// TIA Portal V20 export
FUNCTION_BLOCK "Simulation"   // FB100, LAD
// stored: MemoryReserve 100, Namespace Unit1.Em2, SetENOAutomatically false
   VAR
      Simulation_addon_Instance { S7_SetPoint := 'True'} : "Simulation_addon";
      Simulation_addon_Instance_1 { S7_SetPoint := 'True'} : "Simulation_addon";
      Simulation_addon_Instance_2 { S7_SetPoint := 'True'} : "Simulation_addon";
      Simulation_addon_Instance_3 { S7_SetPoint := 'True'} : "Simulation_addon";
      Simulation_addon_Instance_4 { S7_SetPoint := 'True'} : "Simulation_addon";
      Simulation_addon_Instance_5 { S7_SetPoint := 'True'} : "Simulation_addon";
      Simulation_addon_Instance_6 { S7_SetPoint := 'True'} : "Simulation_addon";
      Simulation_addon_Instance_7 { S7_SetPoint := 'True'} : "Simulation_addon";
      Simulation_addon_Instance_8 { S7_SetPoint := 'True'} : "Simulation_addon";
      Simulation_addon_Instance_9 { S7_SetPoint := 'True'} : "Simulation_addon";
      Simulation_addon_Instance_10 { S7_SetPoint := 'True'} : "Simulation_addon";
      Simulation_addon_Instance_11 { S7_SetPoint := 'True'} : "Simulation_addon";
      Simulation_addon_Instance_12 { S7_SetPoint := 'True'} : "Simulation_addon";
      Simulation_addon_Instance_13 { S7_SetPoint := 'True'} : "Simulation_addon";
      Simulation_addon_Instance_14 { S7_SetPoint := 'True'} : "Simulation_addon";
      Simulation_addon_Instance_15 { S7_SetPoint := 'True'} : "Simulation_addon";
      Simulation_addon_Instance_16 { S7_SetPoint := 'True'} : "Simulation_addon";
      Simulation_addon_Instance_17 { S7_SetPoint := 'True'} : "Simulation_addon";
      Simulation_addon_Instance_18 { S7_SetPoint := 'True'} : "Simulation_addon";
      Simulation_addon_Instance_19 { S7_SetPoint := 'True'} : "Simulation_addon";
      Simulation_addon_Instance_20 { S7_SetPoint := 'True'} : "Simulation_addon";
      Simulation_addon_Instance_21 { S7_SetPoint := 'True'} : "Simulation_addon";
   END_VAR
BEGIN

REGION Network 1: cmElectrodeFixRightTopFwdBwd
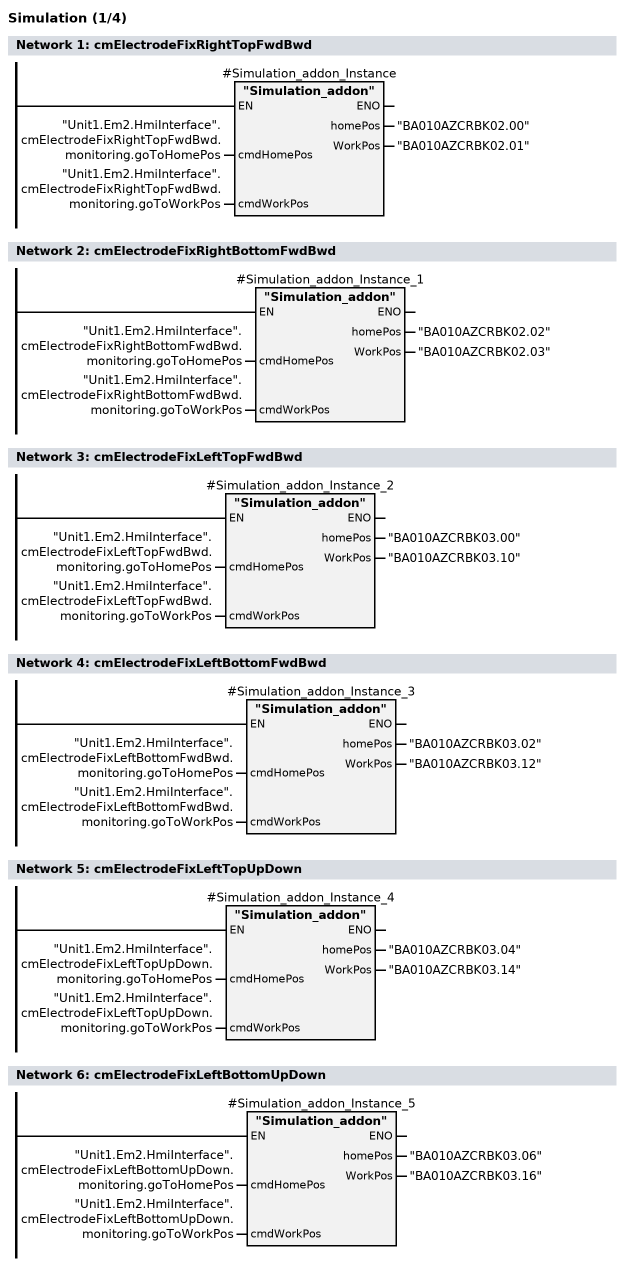
   RUNG wire#powerrail
      #Simulation_addon_Instance(cmdHomePos := "Unit1.Em2.HmiInterface".cmElectrodeFixRightTopFwdBwd.monitoring.goToHomePos, cmdWorkPos := "Unit1.Em2.HmiInterface".cmElectrodeFixRightTopFwdBwd.monitoring.goToWorkPos, homePos => "BA010AZCRBK02.00", WorkPos => "BA010AZCRBK02.01")
   END_RUNG
   // the same network as SCL:
   #Simulation_addon_Instance(cmdHomePos := "Unit1.Em2.HmiInterface".cmElectrodeFixRightTopFwdBwd.monitoring.goToHomePos,   // "Simulation_addon"
                           cmdWorkPos := "Unit1.Em2.HmiInterface".cmElectrodeFixRightTopFwdBwd.monitoring.goToWorkPos,
                           homePos => "BA010AZCRBK02.00",
                           WorkPos => "BA010AZCRBK02.01");
END_REGION

REGION Network 2: cmElectrodeFixRightBottomFwdBwd
   RUNG wire#powerrail
      #Simulation_addon_Instance_1(cmdHomePos := "Unit1.Em2.HmiInterface".cmElectrodeFixRightBottomFwdBwd.monitoring.goToHomePos, cmdWorkPos := "Unit1.Em2.HmiInterface".cmElectrodeFixRightBottomFwdBwd.monitoring.goToWorkPos, homePos => "BA010AZCRBK02.02", WorkPos => "BA010AZCRBK02.03")
   END_RUNG
   // the same network as SCL:
   #Simulation_addon_Instance_1(cmdHomePos := "Unit1.Em2.HmiInterface".cmElectrodeFixRightBottomFwdBwd.monitoring.goToHomePos,   // "Simulation_addon"
                           cmdWorkPos := "Unit1.Em2.HmiInterface".cmElectrodeFixRightBottomFwdBwd.monitoring.goToWorkPos,
                           homePos => "BA010AZCRBK02.02",
                           WorkPos => "BA010AZCRBK02.03");
END_REGION

REGION Network 3: cmElectrodeFixLeftTopFwdBwd
   RUNG wire#powerrail
      #Simulation_addon_Instance_2(cmdHomePos := "Unit1.Em2.HmiInterface".cmElectrodeFixLeftTopFwdBwd.monitoring.goToHomePos, cmdWorkPos := "Unit1.Em2.HmiInterface".cmElectrodeFixLeftTopFwdBwd.monitoring.goToWorkPos, homePos => "BA010AZCRBK03.00", WorkPos => "BA010AZCRBK03.10")
   END_RUNG
   // the same network as SCL:
   #Simulation_addon_Instance_2(cmdHomePos := "Unit1.Em2.HmiInterface".cmElectrodeFixLeftTopFwdBwd.monitoring.goToHomePos,   // "Simulation_addon"
                           cmdWorkPos := "Unit1.Em2.HmiInterface".cmElectrodeFixLeftTopFwdBwd.monitoring.goToWorkPos,
                           homePos => "BA010AZCRBK03.00",
                           WorkPos => "BA010AZCRBK03.10");
END_REGION

REGION Network 4: cmElectrodeFixLeftBottomFwdBwd
   RUNG wire#powerrail
      #Simulation_addon_Instance_3(cmdHomePos := "Unit1.Em2.HmiInterface".cmElectrodeFixLeftBottomFwdBwd.monitoring.goToHomePos, cmdWorkPos := "Unit1.Em2.HmiInterface".cmElectrodeFixLeftBottomFwdBwd.monitoring.goToWorkPos, homePos => "BA010AZCRBK03.02", WorkPos => "BA010AZCRBK03.12")
   END_RUNG
   // the same network as SCL:
   #Simulation_addon_Instance_3(cmdHomePos := "Unit1.Em2.HmiInterface".cmElectrodeFixLeftBottomFwdBwd.monitoring.goToHomePos,   // "Simulation_addon"
                           cmdWorkPos := "Unit1.Em2.HmiInterface".cmElectrodeFixLeftBottomFwdBwd.monitoring.goToWorkPos,
                           homePos => "BA010AZCRBK03.02",
                           WorkPos => "BA010AZCRBK03.12");
END_REGION

REGION Network 5: cmElectrodeFixLeftTopUpDown
   RUNG wire#powerrail
      #Simulation_addon_Instance_4(cmdHomePos := "Unit1.Em2.HmiInterface".cmElectrodeFixLeftTopUpDown.monitoring.goToHomePos, cmdWorkPos := "Unit1.Em2.HmiInterface".cmElectrodeFixLeftTopUpDown.monitoring.goToWorkPos, homePos => "BA010AZCRBK03.04", WorkPos => "BA010AZCRBK03.14")
   END_RUNG
   // the same network as SCL:
   #Simulation_addon_Instance_4(cmdHomePos := "Unit1.Em2.HmiInterface".cmElectrodeFixLeftTopUpDown.monitoring.goToHomePos,   // "Simulation_addon"
                           cmdWorkPos := "Unit1.Em2.HmiInterface".cmElectrodeFixLeftTopUpDown.monitoring.goToWorkPos,
                           homePos => "BA010AZCRBK03.04",
                           WorkPos => "BA010AZCRBK03.14");
END_REGION

REGION Network 6: cmElectrodeFixLeftBottomUpDown
   RUNG wire#powerrail
      #Simulation_addon_Instance_5(cmdHomePos := "Unit1.Em2.HmiInterface".cmElectrodeFixLeftBottomUpDown.monitoring.goToHomePos, cmdWorkPos := "Unit1.Em2.HmiInterface".cmElectrodeFixLeftBottomUpDown.monitoring.goToWorkPos, homePos => "BA010AZCRBK03.06", WorkPos => "BA010AZCRBK03.16")
   END_RUNG
   // the same network as SCL:
   #Simulation_addon_Instance_5(cmdHomePos := "Unit1.Em2.HmiInterface".cmElectrodeFixLeftBottomUpDown.monitoring.goToHomePos,   // "Simulation_addon"
                           cmdWorkPos := "Unit1.Em2.HmiInterface".cmElectrodeFixLeftBottomUpDown.monitoring.goToWorkPos,
                           homePos => "BA010AZCRBK03.06",
                           WorkPos => "BA010AZCRBK03.16");
END_REGION

REGION Network 7: cmUwSemiSplicerVacuumRightTopOnOff
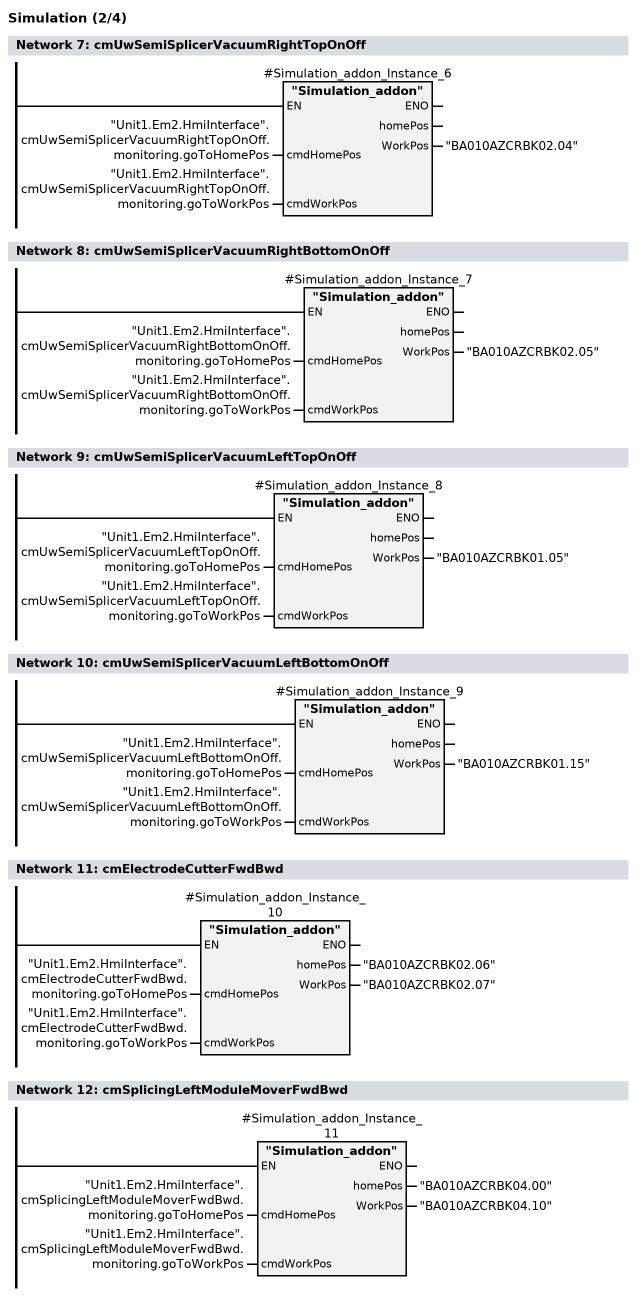
   RUNG wire#powerrail
      #Simulation_addon_Instance_6(cmdHomePos := "Unit1.Em2.HmiInterface".cmUwSemiSplicerVacuumRightTopOnOff.monitoring.goToHomePos, cmdWorkPos := "Unit1.Em2.HmiInterface".cmUwSemiSplicerVacuumRightTopOnOff.monitoring.goToWorkPos, homePos =>, WorkPos => "BA010AZCRBK02.04")
   END_RUNG
   // the same network as SCL:
   #Simulation_addon_Instance_6(cmdHomePos := "Unit1.Em2.HmiInterface".cmUwSemiSplicerVacuumRightTopOnOff.monitoring.goToHomePos,   // "Simulation_addon"
                           cmdWorkPos := "Unit1.Em2.HmiInterface".cmUwSemiSplicerVacuumRightTopOnOff.monitoring.goToWorkPos,
                           WorkPos => "BA010AZCRBK02.04");
END_REGION

REGION Network 8: cmUwSemiSplicerVacuumRightBottomOnOff
   RUNG wire#powerrail
      #Simulation_addon_Instance_7(cmdHomePos := "Unit1.Em2.HmiInterface".cmUwSemiSplicerVacuumRightBottomOnOff.monitoring.goToHomePos, cmdWorkPos := "Unit1.Em2.HmiInterface".cmUwSemiSplicerVacuumRightBottomOnOff.monitoring.goToWorkPos, homePos =>, WorkPos => "BA010AZCRBK02.05")
   END_RUNG
   // the same network as SCL:
   #Simulation_addon_Instance_7(cmdHomePos := "Unit1.Em2.HmiInterface".cmUwSemiSplicerVacuumRightBottomOnOff.monitoring.goToHomePos,   // "Simulation_addon"
                           cmdWorkPos := "Unit1.Em2.HmiInterface".cmUwSemiSplicerVacuumRightBottomOnOff.monitoring.goToWorkPos,
                           WorkPos => "BA010AZCRBK02.05");
END_REGION

REGION Network 9: cmUwSemiSplicerVacuumLeftTopOnOff
   RUNG wire#powerrail
      #Simulation_addon_Instance_8(cmdHomePos := "Unit1.Em2.HmiInterface".cmUwSemiSplicerVacuumLeftTopOnOff.monitoring.goToHomePos, cmdWorkPos := "Unit1.Em2.HmiInterface".cmUwSemiSplicerVacuumLeftTopOnOff.monitoring.goToWorkPos, homePos =>, WorkPos => "BA010AZCRBK01.05")
   END_RUNG
   // the same network as SCL:
   #Simulation_addon_Instance_8(cmdHomePos := "Unit1.Em2.HmiInterface".cmUwSemiSplicerVacuumLeftTopOnOff.monitoring.goToHomePos,   // "Simulation_addon"
                           cmdWorkPos := "Unit1.Em2.HmiInterface".cmUwSemiSplicerVacuumLeftTopOnOff.monitoring.goToWorkPos,
                           WorkPos => "BA010AZCRBK01.05");
END_REGION

REGION Network 10: cmUwSemiSplicerVacuumLeftBottomOnOff
   RUNG wire#powerrail
      #Simulation_addon_Instance_9(cmdHomePos := "Unit1.Em2.HmiInterface".cmUwSemiSplicerVacuumLeftBottomOnOff.monitoring.goToHomePos, cmdWorkPos := "Unit1.Em2.HmiInterface".cmUwSemiSplicerVacuumLeftBottomOnOff.monitoring.goToWorkPos, homePos =>, WorkPos => "BA010AZCRBK01.15")
   END_RUNG
   // the same network as SCL:
   #Simulation_addon_Instance_9(cmdHomePos := "Unit1.Em2.HmiInterface".cmUwSemiSplicerVacuumLeftBottomOnOff.monitoring.goToHomePos,   // "Simulation_addon"
                           cmdWorkPos := "Unit1.Em2.HmiInterface".cmUwSemiSplicerVacuumLeftBottomOnOff.monitoring.goToWorkPos,
                           WorkPos => "BA010AZCRBK01.15");
END_REGION

REGION Network 11: cmElectrodeCutterFwdBwd
   RUNG wire#powerrail
      #Simulation_addon_Instance_10(cmdHomePos := "Unit1.Em2.HmiInterface".cmElectrodeCutterFwdBwd.monitoring.goToHomePos, cmdWorkPos := "Unit1.Em2.HmiInterface".cmElectrodeCutterFwdBwd.monitoring.goToWorkPos, homePos => "BA010AZCRBK02.06", WorkPos => "BA010AZCRBK02.07")
   END_RUNG
   // the same network as SCL:
   #Simulation_addon_Instance_10(cmdHomePos := "Unit1.Em2.HmiInterface".cmElectrodeCutterFwdBwd.monitoring.goToHomePos,   // "Simulation_addon"
                           cmdWorkPos := "Unit1.Em2.HmiInterface".cmElectrodeCutterFwdBwd.monitoring.goToWorkPos,
                           homePos => "BA010AZCRBK02.06",
                           WorkPos => "BA010AZCRBK02.07");
END_REGION

REGION Network 12: cmSplicingLeftModuleMoverFwdBwd
   RUNG wire#powerrail
      #Simulation_addon_Instance_11(cmdHomePos := "Unit1.Em2.HmiInterface".cmSplicingLeftModuleMoverFwdBwd.monitoring.goToHomePos, cmdWorkPos := "Unit1.Em2.HmiInterface".cmSplicingLeftModuleMoverFwdBwd.monitoring.goToWorkPos, homePos => "BA010AZCRBK04.00", WorkPos => "BA010AZCRBK04.10")
   END_RUNG
   // the same network as SCL:
   #Simulation_addon_Instance_11(cmdHomePos := "Unit1.Em2.HmiInterface".cmSplicingLeftModuleMoverFwdBwd.monitoring.goToHomePos,   // "Simulation_addon"
                           cmdWorkPos := "Unit1.Em2.HmiInterface".cmSplicingLeftModuleMoverFwdBwd.monitoring.goToWorkPos,
                           homePos => "BA010AZCRBK04.00",
                           WorkPos => "BA010AZCRBK04.10");
END_REGION

REGION Network 13: cmSplicingRightModuleMoverFwdBwd
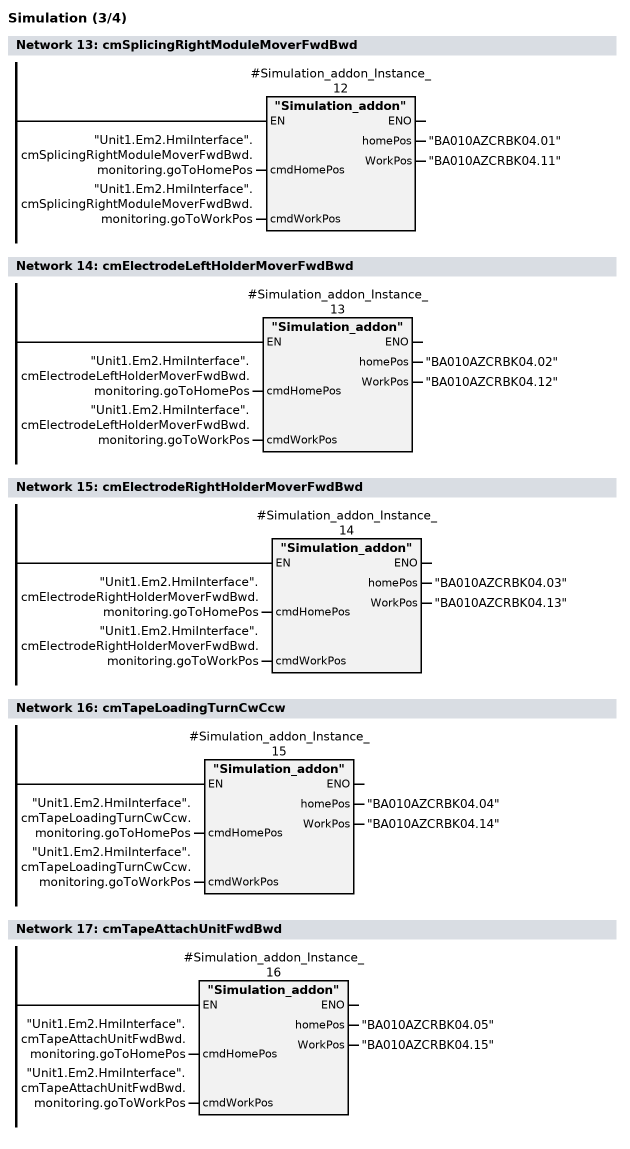
   RUNG wire#powerrail
      #Simulation_addon_Instance_12(cmdHomePos := "Unit1.Em2.HmiInterface".cmSplicingRightModuleMoverFwdBwd.monitoring.goToHomePos, cmdWorkPos := "Unit1.Em2.HmiInterface".cmSplicingRightModuleMoverFwdBwd.monitoring.goToWorkPos, homePos => "BA010AZCRBK04.01", WorkPos => "BA010AZCRBK04.11")
   END_RUNG
   // the same network as SCL:
   #Simulation_addon_Instance_12(cmdHomePos := "Unit1.Em2.HmiInterface".cmSplicingRightModuleMoverFwdBwd.monitoring.goToHomePos,   // "Simulation_addon"
                           cmdWorkPos := "Unit1.Em2.HmiInterface".cmSplicingRightModuleMoverFwdBwd.monitoring.goToWorkPos,
                           homePos => "BA010AZCRBK04.01",
                           WorkPos => "BA010AZCRBK04.11");
END_REGION

REGION Network 14: cmElectrodeLeftHolderMoverFwdBwd
   RUNG wire#powerrail
      #Simulation_addon_Instance_13(cmdHomePos := "Unit1.Em2.HmiInterface".cmElectrodeLeftHolderMoverFwdBwd.monitoring.goToHomePos, cmdWorkPos := "Unit1.Em2.HmiInterface".cmElectrodeLeftHolderMoverFwdBwd.monitoring.goToWorkPos, homePos => "BA010AZCRBK04.02", WorkPos => "BA010AZCRBK04.12")
   END_RUNG
   // the same network as SCL:
   #Simulation_addon_Instance_13(cmdHomePos := "Unit1.Em2.HmiInterface".cmElectrodeLeftHolderMoverFwdBwd.monitoring.goToHomePos,   // "Simulation_addon"
                           cmdWorkPos := "Unit1.Em2.HmiInterface".cmElectrodeLeftHolderMoverFwdBwd.monitoring.goToWorkPos,
                           homePos => "BA010AZCRBK04.02",
                           WorkPos => "BA010AZCRBK04.12");
END_REGION

REGION Network 15: cmElectrodeRightHolderMoverFwdBwd
   RUNG wire#powerrail
      #Simulation_addon_Instance_14(cmdHomePos := "Unit1.Em2.HmiInterface".cmElectrodeRightHolderMoverFwdBwd.monitoring.goToHomePos, cmdWorkPos := "Unit1.Em2.HmiInterface".cmElectrodeRightHolderMoverFwdBwd.monitoring.goToWorkPos, homePos => "BA010AZCRBK04.03", WorkPos => "BA010AZCRBK04.13")
   END_RUNG
   // the same network as SCL:
   #Simulation_addon_Instance_14(cmdHomePos := "Unit1.Em2.HmiInterface".cmElectrodeRightHolderMoverFwdBwd.monitoring.goToHomePos,   // "Simulation_addon"
                           cmdWorkPos := "Unit1.Em2.HmiInterface".cmElectrodeRightHolderMoverFwdBwd.monitoring.goToWorkPos,
                           homePos => "BA010AZCRBK04.03",
                           WorkPos => "BA010AZCRBK04.13");
END_REGION

REGION Network 16: cmTapeLoadingTurnCwCcw
   RUNG wire#powerrail
      #Simulation_addon_Instance_15(cmdHomePos := "Unit1.Em2.HmiInterface".cmTapeLoadingTurnCwCcw.monitoring.goToHomePos, cmdWorkPos := "Unit1.Em2.HmiInterface".cmTapeLoadingTurnCwCcw.monitoring.goToWorkPos, homePos => "BA010AZCRBK04.04", WorkPos => "BA010AZCRBK04.14")
   END_RUNG
   // the same network as SCL:
   #Simulation_addon_Instance_15(cmdHomePos := "Unit1.Em2.HmiInterface".cmTapeLoadingTurnCwCcw.monitoring.goToHomePos,   // "Simulation_addon"
                           cmdWorkPos := "Unit1.Em2.HmiInterface".cmTapeLoadingTurnCwCcw.monitoring.goToWorkPos,
                           homePos => "BA010AZCRBK04.04",
                           WorkPos => "BA010AZCRBK04.14");
END_REGION

REGION Network 17: cmTapeAttachUnitFwdBwd
   RUNG wire#powerrail
      #Simulation_addon_Instance_16(cmdHomePos := "Unit1.Em2.HmiInterface".cmTapeAttachUnitFwdBwd.monitoring.goToHomePos, cmdWorkPos := "Unit1.Em2.HmiInterface".cmTapeAttachUnitFwdBwd.monitoring.goToWorkPos, homePos => "BA010AZCRBK04.05", WorkPos => "BA010AZCRBK04.15")
   END_RUNG
   // the same network as SCL:
   #Simulation_addon_Instance_16(cmdHomePos := "Unit1.Em2.HmiInterface".cmTapeAttachUnitFwdBwd.monitoring.goToHomePos,   // "Simulation_addon"
                           cmdWorkPos := "Unit1.Em2.HmiInterface".cmTapeAttachUnitFwdBwd.monitoring.goToWorkPos,
                           homePos => "BA010AZCRBK04.05",
                           WorkPos => "BA010AZCRBK04.15");
END_REGION

REGION Network 18: SemiSplicerTapeVacuumOnOff
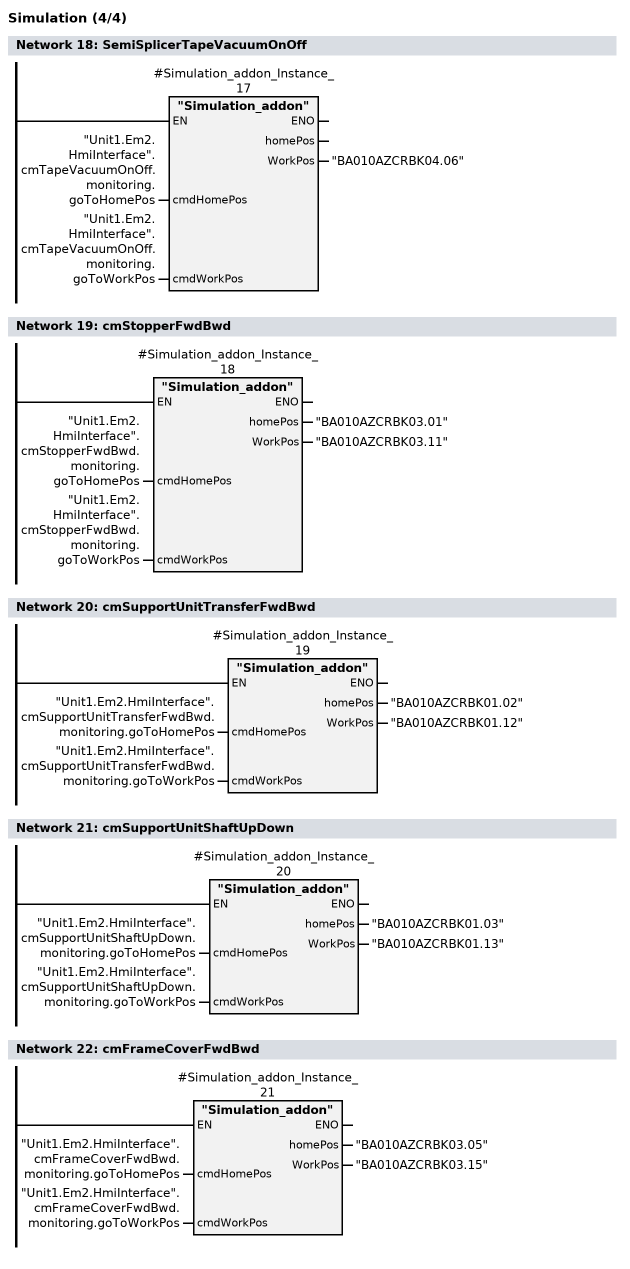
   RUNG wire#powerrail
      #Simulation_addon_Instance_17(cmdHomePos := "Unit1.Em2.HmiInterface".cmTapeVacuumOnOff.monitoring.goToHomePos, cmdWorkPos := "Unit1.Em2.HmiInterface".cmTapeVacuumOnOff.monitoring.goToWorkPos, homePos =>, WorkPos => "BA010AZCRBK04.06")
   END_RUNG
   // the same network as SCL:
   #Simulation_addon_Instance_17(cmdHomePos := "Unit1.Em2.HmiInterface".cmTapeVacuumOnOff.monitoring.goToHomePos,   // "Simulation_addon"
                           cmdWorkPos := "Unit1.Em2.HmiInterface".cmTapeVacuumOnOff.monitoring.goToWorkPos,
                           WorkPos => "BA010AZCRBK04.06");
END_REGION

REGION Network 19: cmStopperFwdBwd
   RUNG wire#powerrail
      #Simulation_addon_Instance_18(cmdHomePos := "Unit1.Em2.HmiInterface".cmStopperFwdBwd.monitoring.goToHomePos, cmdWorkPos := "Unit1.Em2.HmiInterface".cmStopperFwdBwd.monitoring.goToWorkPos, homePos => "BA010AZCRBK03.01", WorkPos => "BA010AZCRBK03.11")
   END_RUNG
   // the same network as SCL:
   #Simulation_addon_Instance_18(cmdHomePos := "Unit1.Em2.HmiInterface".cmStopperFwdBwd.monitoring.goToHomePos,   // "Simulation_addon"
                           cmdWorkPos := "Unit1.Em2.HmiInterface".cmStopperFwdBwd.monitoring.goToWorkPos,
                           homePos => "BA010AZCRBK03.01",
                           WorkPos => "BA010AZCRBK03.11");
END_REGION

REGION Network 20: cmSupportUnitTransferFwdBwd
   RUNG wire#powerrail
      #Simulation_addon_Instance_19(cmdHomePos := "Unit1.Em2.HmiInterface".cmSupportUnitTransferFwdBwd.monitoring.goToHomePos, cmdWorkPos := "Unit1.Em2.HmiInterface".cmSupportUnitTransferFwdBwd.monitoring.goToWorkPos, homePos => "BA010AZCRBK01.02", WorkPos => "BA010AZCRBK01.12")
   END_RUNG
   // the same network as SCL:
   #Simulation_addon_Instance_19(cmdHomePos := "Unit1.Em2.HmiInterface".cmSupportUnitTransferFwdBwd.monitoring.goToHomePos,   // "Simulation_addon"
                           cmdWorkPos := "Unit1.Em2.HmiInterface".cmSupportUnitTransferFwdBwd.monitoring.goToWorkPos,
                           homePos => "BA010AZCRBK01.02",
                           WorkPos => "BA010AZCRBK01.12");
END_REGION

REGION Network 21: cmSupportUnitShaftUpDown
   RUNG wire#powerrail
      #Simulation_addon_Instance_20(cmdHomePos := "Unit1.Em2.HmiInterface".cmSupportUnitShaftUpDown.monitoring.goToHomePos, cmdWorkPos := "Unit1.Em2.HmiInterface".cmSupportUnitShaftUpDown.monitoring.goToWorkPos, homePos => "BA010AZCRBK01.03", WorkPos => "BA010AZCRBK01.13")
   END_RUNG
   // the same network as SCL:
   #Simulation_addon_Instance_20(cmdHomePos := "Unit1.Em2.HmiInterface".cmSupportUnitShaftUpDown.monitoring.goToHomePos,   // "Simulation_addon"
                           cmdWorkPos := "Unit1.Em2.HmiInterface".cmSupportUnitShaftUpDown.monitoring.goToWorkPos,
                           homePos => "BA010AZCRBK01.03",
                           WorkPos => "BA010AZCRBK01.13");
END_REGION

REGION Network 22: cmFrameCoverFwdBwd
   RUNG wire#powerrail
      #Simulation_addon_Instance_21(cmdHomePos := "Unit1.Em2.HmiInterface".cmFrameCoverFwdBwd.monitoring.goToHomePos, cmdWorkPos := "Unit1.Em2.HmiInterface".cmFrameCoverFwdBwd.monitoring.goToWorkPos, homePos => "BA010AZCRBK03.05", WorkPos => "BA010AZCRBK03.15")
   END_RUNG
   // the same network as SCL:
   #Simulation_addon_Instance_21(cmdHomePos := "Unit1.Em2.HmiInterface".cmFrameCoverFwdBwd.monitoring.goToHomePos,   // "Simulation_addon"
                           cmdWorkPos := "Unit1.Em2.HmiInterface".cmFrameCoverFwdBwd.monitoring.goToWorkPos,
                           homePos => "BA010AZCRBK03.05",
                           WorkPos => "BA010AZCRBK03.15");
END_REGION
END_FUNCTION_BLOCK
